# EPICS IOC start-up script: iocBoot/ioc6idACS1/settings.iocsh
# Shell prompt
epicsEnvSet("IOCSH_PS1", "$(IOC)> ")

# prefix used for all PVs in this IOC
epicsEnvSet("PREFIX", "6idACS1:")

#For devIocStats
epicsEnvSet("ENGINEER", "engineer")
epicsEnvSet("LOCATION", "location")
epicsEnvSet("GROUP", "group")

# search path for database files
epicsEnvSet("EPICS_DB_INCLUDE_PATH", ".")

# search path for streamDevice protocol files
epicsEnvSet("STREAM_PROTOCOL_PATH", ".")

# search path for lua scripts
# epicsEnvSet("LUA_SCRIPT_PATH", "./scripts")

# Specify largest array CA will transport
# Note for N doubles, need N*8 bytes+some overhead
epicsEnvSet("EPICS_CA_MAX_ARRAY_BYTES", 64010)
